TYPE ST_MESSAGE_CTRL :
STRUCT
  Cmd         : E_MESSAGE_CTRL;
END_STRUCT
END_TYPE

(* stored: Version 1.1.0.1
   DUT ST_MESSAGE_CTRL: Id {c0a0c942-c33b-4b1c-91b6-3018de854c3c} *)
